Staubli VAL3: listframe.pgx

program listframe(string pTitle (dimensions=1), num pX (dimensions=1), num pY (dimensions=1), num pDx (dimensions=1), num pDy (dimensions=1))
  local num lDx
  local num lDy
  local num lI
  local num lJ
  local string lStr
  local string lStrLine
  local num lValue
begin
  //
  // Staubli Copyright 2003 06 20
  //
  lStrLine="─────────────────────────────────────────"
  lDx=pDx
  lDy=pDy
  //Top
  lStr="┌"+mid(lStrLine,lDx,0)+"┐"
  gotoxy(pX,pY)
  put(lStr)
  lValue=pX+2
  //Title
  if pTitle!=""
    call leftPos("┤"+pTitle+"├",lDx,pTitle)
    gotoxy(pX+lDx-getDisplayLen(pTitle)+1,pY)
    put(pTitle)
  endIf
  //Containt
  for lJ=1 to lDy
    lValue=pY+lJ
    lStr="│"
    gotoxy(pX,lValue)
    put(lStr)
    gotoxy(pX+lDx+1,lValue)
    put(lStr)
  endFor
  //Bottom
  lValue=pY+lJ
  lStr="└"+mid(lStrLine,lDx,0)+"┘"
  gotoxy(pX,lValue)
  put(lStr)
end
